// Mitsubishi GX Works2 project: BookEX5_0 ST   PLC: Q13UDV

TYPE DateTime : STRUCT
  Year : INT;
  Month : INT;
  Day : INT;
  WeekDay : INT;
  iHour : INT;
  iMin : INT;
  iSec : INT;
  ms : INT;
END_STRUCT END_TYPE

TYPE Vector : STRUCT
  axisX : REAL;
  axisY : REAL;
  axisZ : REAL;
END_STRUCT END_TYPE

TYPE WordBit : STRUCT
  Data : DWORD;
  Flag : BOOL;
END_STRUCT END_TYPE

// global labels: Global
VAR_GLOBAL
  bVar0 AT M5000 : BOOL;
  abArray0 AT M5010 : ARRAY [0..49] OF BOOL;
  sStr0 AT D5000 : STRING[199];
  sStr1 AT D5100 : STRING[199];
  sStr2 AT D5200 : STRING[199];
  sStr3 AT D5300 : STRING[199];
  sStr4 AT D5400 : STRING[199];
  sStr5 AT D5500 : STRING[199];
  sStr6 AT D5600 : STRING[199];
  sStr7 AT D5700 : STRING[199];
  sStr8 AT D5800 : STRING[199];
  sStr9 AT D5900 : STRING[199];
  iVar0 AT D4500 : INT;
  iVar1 AT D4501 : INT;
  iVar2 AT D4502 : INT;
  iVar3 AT D4503 : INT;
  iVar4 AT D4504 : INT;
  iVar5 AT D4505 : INT;
  iVar6 AT D4506 : INT;
  iVar7 AT D4507 : INT;
  iVar8 AT D4508 : INT;
  iVar9 AT D4509 : INT;
  dVar0 AT D4510 : DINT;
  dVar1 AT D4512 : DINT;
  dVar2 AT D4514 : DINT;
  dVar3 AT D4516 : DINT;
  dVar4 AT D4518 : DINT;
  dVar5 AT D4520 : DINT;
  dVar6 AT D4522 : DINT;
  dVar7 AT D4524 : DINT;
  dVar8 AT D4526 : DINT;
  dVar9 AT D4528 : DINT;
  wVar0 AT D4530 : WORD;
  wVar1 AT D4531 : WORD;
  wVar2 AT D4532 : WORD;
  wVar3 AT D4533 : WORD;
  wVar4 AT D4534 : WORD;
  wVar5 AT D4535 : WORD;
  wVar6 AT D4536 : WORD;
  wVar7 AT D4537 : WORD;
  wVar8 AT D4538 : WORD;
  wVar9 AT D4539 : WORD;
  dwVar0 AT D4540 : DWORD;
  dwVar1 AT D4542 : DWORD;
  dwVar2 AT D4544 : DWORD;
  dwVar3 AT D4546 : DWORD;
  dwVar4 AT D4548 : DWORD;
  dwVar5 AT D4550 : DWORD;
  dwVar6 AT D4552 : DWORD;
  dwVar7 AT D4554 : DWORD;
  dwVar8 AT D4556 : DWORD;
  dwVar9 AT D4558 : DWORD;
  fsVar0 AT D4560 : REAL;
  fsVar1 AT D4562 : REAL;
  fsVar2 AT D4564 : REAL;
  fsVar3 AT D4566 : REAL;
  fsVar4 AT D4568 : REAL;
  fsVar5 AT D4570 : REAL;
  fsVar6 AT D4572 : REAL;
  fsVar7 AT D4574 : REAL;
  fsVar8 AT D4576 : REAL;
  fsVar9 AT D4578 : REAL;
  fdVar0 AT D4580 : LREAL;
  tTime0 AT D4620 : TIME;
  tTime1 AT D4622 : TIME;
  tTime2 AT D4624 : TIME;
  tTime3 AT D4626 : TIME;
  tTime4 AT D4628 : TIME;
  tTime5 AT D4630 : TIME;
  tTime6 AT D4632 : TIME;
  tTime7 AT D4634 : TIME;
  tTime8 AT D4636 : TIME;
  tTime9 AT D4638 : TIME;
  tTime10 AT D4640 : TIME;
  bVar1 AT M5001 : BOOL;
  bVar2 AT M5002 : BOOL;
  bVar3 AT M5003 : BOOL;
  bVar4 AT M5004 : BOOL;
  bVar5 AT M5005 : BOOL;
  bVar6 AT M5006 : BOOL;
  bVar7 AT M5007 : BOOL;
  bVar8 AT M5008 : BOOL;
  bVar9 AT M5009 : BOOL;
  abArray1 AT M5060 : ARRAY [0..49] OF BOOL;
  abArray2 AT M5110 : ARRAY [0..49] OF BOOL;
  abArray3 AT M5160 : ARRAY [0..49] OF BOOL;
  abArray4 AT M5210 : ARRAY [0..49] OF BOOL;
  abArray5 AT M5260 : ARRAY [0..49] OF BOOL;
  abArray6 AT M5310 : ARRAY [0..49] OF BOOL;
  abArray7 AT M5360 : ARRAY [0..49] OF BOOL;
  abArray8 AT M5410 : ARRAY [0..49] OF BOOL;
  abArray9 AT M5460 : ARRAY [0..49] OF BOOL;
  fdVar1 AT D4584 : LREAL;
  fdVar2 AT D4588 : LREAL;
  fdVar3 AT D4592 : LREAL;
  fdVar4 AT D4596 : LREAL;
  fdVar5 AT D4600 : LREAL;
  fdVar6 AT D4604 : LREAL;
  fdVar7 AT D4608 : LREAL;
  fdVar8 AT D4612 : LREAL;
  fdVar9 AT D4616 : LREAL;
  aSendData1 AT D100 : ARRAY [0..9] OF INT;
  aRecvData1 AT D110 : ARRAY [0..9] OF INT;
  aSendData2 AT D120 : ARRAY [0..9] OF INT;
  aRecvData2 AT D130 : ARRAY [0..9] OF INT;
END_VAR
// user libraries (not included): HMI

FUNCTION_BLOCK AllFB
VAR_INPUT
  b_IN1 : BOOL;
  b_IN2 : BOOL;
END_VAR
VAR_OUTPUT
  b_OT : BOOL;
END_VAR
(* structured ladder/FBD written out as ST: instructions are called as NAME(EN, inputs, outputs); _pN, _eN, _tN stand for wires *)
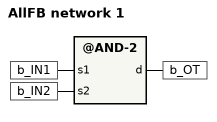
(* network 1 *)
b_OT := @AND-2(b_IN1, b_IN2);
END_FUNCTION_BLOCK

FUNCTION_BLOCK EnFB
VAR_INPUT
  b_IN1 : BOOL;
  b_IN2 : BOOL;
END_VAR
VAR_OUTPUT
  b_OT : BOOL;
END_VAR
(* structured ladder/FBD written out as ST: instructions are called as NAME(EN, inputs, outputs); _pN, _eN, _tN stand for wires *)
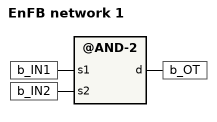
(* network 1 *)
b_OT := @AND-2(b_IN1, b_IN2);
END_FUNCTION_BLOCK

FUNCTION EnFUN
VAR_INPUT
  b_IN1 : BOOL;
  b_IN2 : BOOL;
END_VAR
(* structured ladder/FBD written out as ST: instructions are called as NAME(EN, inputs, outputs); _pN, _eN, _tN stand for wires *)
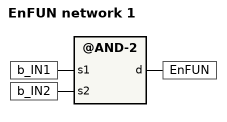
(* network 1 *)
EnFUN := @AND-2(b_IN1, b_IN2);
END_FUNCTION

FUNCTION_BLOCK MacroEnFB
VAR_INPUT
  b_IN1 : BOOL;
  b_IN2 : BOOL;
END_VAR
VAR_OUTPUT
  b_OT : BOOL;
END_VAR
(* structured ladder/FBD written out as ST: instructions are called as NAME(EN, inputs, outputs); _pN, _eN, _tN stand for wires *)
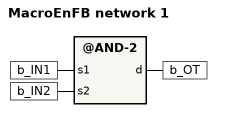
(* network 1 *)
b_OT := @AND-2(b_IN1, b_IN2);
END_FUNCTION_BLOCK

FUNCTION_BLOCK MacroFB
VAR_INPUT
  b_IN1 : BOOL;
  b_IN2 : BOOL;
END_VAR
VAR_OUTPUT
  b_OT : BOOL;
END_VAR
VAR
  ix : INT;
END_VAR
(* structured ladder/FBD written out as ST: instructions are called as NAME(EN, inputs, outputs); _pN, _eN, _tN stand for wires *)
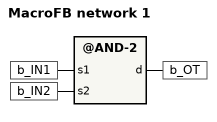
(* network 1 *)
b_OT := @AND-2(b_IN1, b_IN2);
END_FUNCTION_BLOCK

FUNCTION_BLOCK ManEnFB
VAR_INPUT
  b_EN : BOOL;
  b_IN2 : BOOL;
END_VAR
VAR_OUTPUT
  b_OT : BOOL;
END_VAR
VAR
  ix : INT;
END_VAR
VAR_INPUT
  b_IN1 : BOOL;
END_VAR
VAR_OUTPUT
  b_ENO : BOOL;
END_VAR
(* structured ladder/FBD written out as ST: instructions are called as NAME(EN, inputs, outputs); _pN, _eN, _tN stand for wires *)
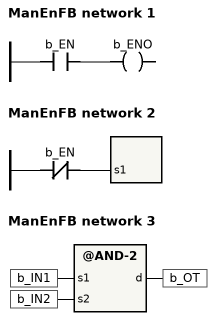
(* network 1 *)
b_ENO := b_EN;
(* network 2 *)
(* element kind 10  <- NOT b_EN *)
(* network 3 *)
b_OT := @AND-2(b_IN1, b_IN2);
END_FUNCTION_BLOCK

FUNCTION_BLOCK NoneFB
VAR_INPUT
  b_IN1 : BOOL;
  b_IN2 : BOOL;
END_VAR
VAR_OUTPUT
  b_OT : BOOL;
END_VAR
(* structured ladder/FBD written out as ST: instructions are called as NAME(EN, inputs, outputs); _pN, _eN, _tN stand for wires *)
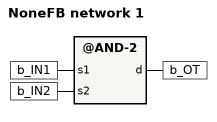
(* network 1 *)
b_OT := @AND-2(b_IN1, b_IN2);
END_FUNCTION_BLOCK

FUNCTION NoneFUN
VAR_INPUT
  b_IN1 : BOOL;
  b_IN2 : BOOL;
END_VAR
(* structured ladder/FBD written out as ST: instructions are called as NAME(EN, inputs, outputs); _pN, _eN, _tN stand for wires *)
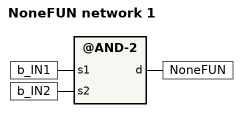
(* network 1 *)
NoneFUN := @AND-2(b_IN1, b_IN2);
END_FUNCTION

PROGRAM 000DataType
VAR
  aBoxNo : ARRAY [0..99] OF INT;
  aStr : ARRAY [0..9] OF STRING[4] := [10('')];
  aStr2 : ARRAY [0..19] OF STRING[32] := [20('')];
  ai박스3 : ARRAY [0..4,0..3,0..2] OF INT;
  aiBox1 : ARRAY [0..4] OF INT;
  aiBox2 : ARRAY [1..5] OF INT;
  ai박스2 : ARRAY [-1..4,1..3] OF INT;
  ix : INT;
  Val1 : INT;
  Val2 : INT;
  Val3 : INT;
  abLable2 : ARRAY [0..4,0..3] OF BOOL;
  abLable1 : ARRAY [0..3] OF BOOL;
  abLabel3 : ARRAY [0..5,0..4,0..3] OF BOOL;
END_VAR
 
FOR ix := 0 TO 99 DO
	aBoxNo[ix] := ix;
END_FOR;
aiBox1[0] := 12;
aiBox1[2] := 34;
aStr[0] := 'ABCDEFG';		(* No Error *)
aStr[1] := '12345678';		(* No Error *)
Val2 := ai박스2[1,1]; 	 
Val3 := 100;
aBoxNo[Val3] := 100;		(* No Error *)
aBoxNo[aBoxNo[aBoxNo[aBoxNo[aBoxNo[Val3]]]]] := 100;
aiBox2 := aiBox1;

Val1 := aBoxNo[55];

bVar0 	:= 1;
bVar1	:= TRUE;
fsVar5	:= E1.0E-5;
fsVar6	:= 1.0E-5;
wVar0	:= 16#FF_FF;
wVar1	:= HFFFF;
aStr2[0]:= 'APP';
aStr2[1]:= '$$';
aStr2[2]:= "$N";
aStr2[3]:= "$n";
aStr2[4]:= "$5C";

MOVP(X1, K3M0, iVar1);

MOVP(X1, K3M0, D40);

DMOVP(X1, 155, dVar0);

DMOVP(X1, 155, D12);

EMOVP(X1, fsVar0, fsVar1);

EDMOVP(X1, 1.23456, fdVar0);
END_PROGRAM

PROGRAM ExCallFB
VAR
  TON_E_1 : TON_E;
  TON_E_2 : TON_E;
  TON_E_3 : TON_E;
  TON_E_4 : TON_E;
END_VAR
 
iVar4 := iVar4 + 1;

TON_E_1.IN := FALSE;
TON_E_1.PT := T#1s;
TON_E_1(EN:=TRUE, IN:=M1);
IF TON_E_1.Q THEN
	TON_E_1(EN:=TRUE, IN:=FALSE);
	iVar1 := iVar1 + 1;
END_IF;
tTime1 := TON_E_1.ET;

TON_E_2(EN:=TRUE, IN:=M1, PT:= T#2s);
IF TON_E_2.Q THEN
	TON_E_2(EN:=TRUE, IN:=FALSE);
	iVar2 := iVar2 + 1;
END_IF;
tTime2 := TON_E_2.ET;

TON_E_3.IN := M1;
TON_E_3.PT := T#3s;
TON_E_3(EN:=TRUE);
IF TON_E_3.Q THEN
	TON_E_3(EN:=TRUE, IN:=FALSE);
	iVar3 := iVar3 + 1;
END_IF;
tTime3 := TON_E_3.ET;

TON_E_4(EN:=TRUE, IN:=M1, PT:= T#2s);
M4 := TON_E_4.Q;
tTime4 := TON_E_4.ET;
IF M4 THEN
	TON_E_4(EN:=TRUE, IN:=FALSE);
	iVar4 := iVar4 + 1;
END_IF;
END_PROGRAM

PROGRAM ExFB
VAR
  NoneFB_1 : NoneFB;
  EnFB_1 : EnFB;
  MacroFB_1 : MacroFB;
  AllFB_1 : AllFB;
  MacroEnFB_1 : MacroEnFB;
  ManEnFB_1 : ManEnFB;
END_VAR
(* structured ladder/FBD written out as ST: instructions are called as NAME(EN, inputs, outputs); _pN, _eN, _tN stand for wires *)
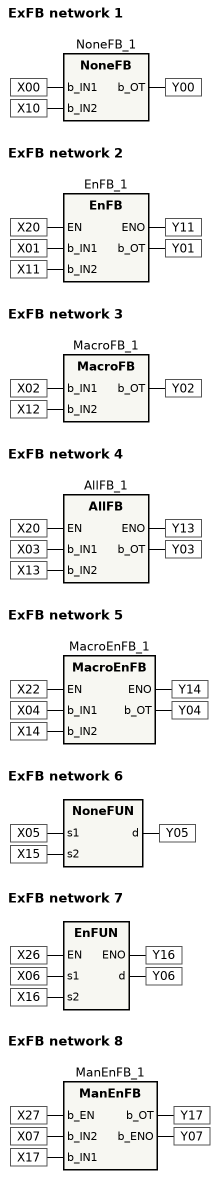
(* network 1 *)
NoneFB_1(b_IN1 := X00, b_IN2 := X10, b_OT => Y00);
(* network 2 *)
EnFB_1(EN := X20, b_IN1 := X01, b_IN2 := X11, ENO => Y11, b_OT => Y01);
(* network 3 *)
MacroFB_1(b_IN1 := X02, b_IN2 := X12, b_OT => Y02);
(* network 4 *)
AllFB_1(EN := X20, b_IN1 := X03, b_IN2 := X13, ENO => Y13, b_OT => Y03);
(* network 5 *)
MacroEnFB_1(EN := X22, b_IN1 := X04, b_IN2 := X14, ENO => Y14, b_OT => Y04);
(* network 6 *)
Y05 := NoneFUN(X05, X15);
(* network 7 *)
_e1 := EnFUN(X26, X06, X16, Y06);
Y16 := _e1;
(* network 8 *)
ManEnFB_1(b_EN := X27, b_IN2 := X07, b_IN1 := X17, b_OT => Y17, b_ENO => Y07);
END_PROGRAM

PROGRAM ExFOR
VAR
  Result1 : BOOL;
  Result2 : BOOL;
END_VAR

iVar4 := 0;
FOR iVar3 := 1 TO 10 BY 1 DO 
	iVar4 := iVar3+iVar4;
END_FOR;

iVar6 := 0;
FOR iVar5 := 10 TO 1 BY -1 DO 
	iVar6 := iVar5+iVar6;
END_FOR;
END_PROGRAM

PROGRAM ExOperator
;
(*기본 연산자*)
iVar0 := iVar1 * iVar2 + iVar3 MOD 16;							(* INT *)
iVar4 := (iVar5 + D0 + iVar6) / 3;
(* iVar0 := dVar1 * iVar2 + iVar3 MOD 16;  데이터형이 틀리면 에러 *)

D0 := iVar1 * D2 + iVar3 MOD 16;
D0 := D1 * (D2+3) / 100;
(* D0 := dVar1 * dVar2 + dVar3 MOD 16;   D0는 INT로 처리함으로 에러 *)

dVar0 := dVar1 * dVar2 / 4 + dVar3 MOD 16;					(* DINT *)
dVar4 := dVar5 / H1000;
(*wVar0 := wVar1 * wVar2 + wVar3 MOD 16;  Bit-string은 일반 연산자 사용시 에러 *)

fsVar0 := fsVar1 + fsVar3 * 2.0;												(* REAL *)
fsVar1 := 2.0  * 3.14 * fsVar5;
fdVar0 := fdVar1 + fdVar2 ** 2.0;

(* sStr0 := sStr0 + "ABC";							String은 일반 연산자 사용시 에러 *)
tTime0 := tTime1+tTime2;															(* Time *)
tTime3 := tTime4 + T#1s;

(*고급 연산자*)
iVar0 := ABS(iVar2 - iVar3);														(* INT *)
dVar0 := ABS(dVar2 - dVar3);													(* DINT *)

fsVar0 := ABS(fsVar1 - fsVar2) + INT_TO_REAL(iVar0);	(* REAL *)
bVar0 := SIN_E (TRUE, fdVar1, fdVar0);
fdVar2 := SQRT((fdVar0 ** 2.0) + (fdVar1 ** 2.0));

(*논리 연산자 *)
bVar0 := bVar1 XOR M0 AND (iVar0 = 100);								(* Bit *)
D1.3 := NOT ( bVar3 AND bVar4);

D0 := D1 AND D2;																				(* WORD *)
wVar1 := wVar1 XOR wVar2;
wVar3 := wVar4 OR H0011;
D3 := D2 OR wVar1;
(* D3 := D2 OR iVar1;  D0는 WORD로  처리함으로 에러 *)

dwVar1 := dwVar1 XOR dwVar2;													(* DWORD *)
dwVar3 := NOT (dwVar4 OR dwVar1) AND H0F0F0F0F;
(* D3 := D2 OR dwVar1;  D0는 WORD로  처리함으로 에러 *)

(*관계연산자*)
bVar0 := bVar1 < bVar2;																	(* Bit *)
bVar0 := ( D0 > 100 ) AND (D0 < 200);											(* INT *)
bVar3 := dVar1 >= 100;																	(* DINT *)
bVar4 := (wVar0 AND H00FF) = 0;												(* WORD *)
bVar4 := wVar1 = H0100;
bVar4 := wVar2 > H0100;
bVar5 := (dwVar0 AND H00FF) <> 0;											(* DWORD *)
bVar6 := dwVar1 <> HFFFFFFFF;
IF D0 = 100 THEN bVar1 := TRUE; ELSE bVar1 := FALSE; END_IF;
bVar7 := tTime0 < tTime1;																(* Time *)
bVar7 := tTime2 > T#200s;
END_PROGRAM

PROGRAM ExREPEAT
VAR
  Result1 : BOOL;
  Result2 : BOOL;
END_VAR

iVar6 := 0;
iVar5 := 1;
REPEAT
	iVar6 := iVar5 + iVar6;
	iVar5 := iVar5 + 1;
	UNTIL iVar5 > 10  
END_REPEAT;
END_PROGRAM

PROGRAM ExST
VAR
  ix : INT;
END_VAR
VAR CONSTANT
  MaxCnt : INT := 100;
END_VAR
VAR
  aaa : ARRAY [0..4,0..4,0..4] OF INT;
  aDT0 : ARRAY [0..2] OF DateTime;
  aDT1 : ARRAY [0..2] OF DateTime;
  DT0 : DateTime;
  DT1 : DateTime;
  aiClass1 : ARRAY [0..9] OF INT;
  aiClass2 : ARRAY [0..9] OF INT;
  Res1 : INT;
  Res2 : INT;
  Res3 : INT;
  Res4 : INT;
END_VAR

(* ST 샘플 츠로그램 *)
wVar1	:= H1234;
dwVar1	:= 12345678;

bVar1	:= BCD_TO_DINT_E(TRUE, wVar1, dVar1);
dVar2	:= BCD_TO_DINT(wVar1);

bVar2	:= ADD_E(TRUE, iVar1, iVar2, iVar3, iVar4, iVar5);
iVar5		:= iVar1 + iVar2 + iVar3 + iVar4;

IF NOT (bVar1 AND NOT bVar2 AND M0) THEN
	bVar2	:= TRUE;
ELSE
	bVar2	:= FALSE;
END_IF;

fbDispHMI(Bit0 := bVar1, Bit1 := bVar2); (* HMI표시를 위한 함수 *)
bVar4	:= fbDispHMI.Data0;


iVar0		:= D10 - 123;

IF iVar0 > 0 THEN
	bVar0	:= TRUE;
ELSE
	bVar1	:= FALSE;
END_IF;

WHILE FunPOU(iVar0) DO
	iVar0		:= iVar0 - 1;
END_WHILE;

bFlag 	:= FunPOU(iVar0 + 1);
fbPOU_1(In0 := iVar0 + 1, Out0 := iVar1);



WHILE bVar0 DO
	iVar0		:= iVar0 - 1;
	IF iVar0 > 100 THEN
		bVar0	:= TRUE;
	ELSE
		IF iVar0 > 50 THEN
			iVar1	:= iVar1 + 1;
		END_IF;
	END_IF;
END_WHILE;




(* 대입문*)
iVar1 			:= iVar2;					iVar3 := 0;
iVar4 			:= iVar4 + 1;
D1 				:= iVar1;
wVar2 		:= INT_TO_WORD(iVar3);
sStr1 			:= 'abc';
sStr2			:= "Apple";

IF LDP(TRUE, M0) THEN
	iVar5 := aiClass2[3];
	iVar7 := DT1.Month;
	aiClass1[3] := 3;
	aDT0[1].Month := 12;
	aiClass2 := aiClass1;
	DT1 := aDT0[1];
	iVar6 := aiClass2[3];
	iVar8 := DT1.Month;
END_IF;

(* IF ... THEN *)
IF M0 THEN
	Y0 := TRUE;
END_IF;

(* IF ... ELSE *)
IF M0 THEN
	Y0 := TRUE;
ELSE
	Y0 := FALSE;
END_IF;

(* IF ... ELSIF *)
IF M0 THEN
	Y0 := TRUE;
ELSIF M1 THEN
	Y1 := TRUE;
ELSIF M2 THEN
	Y2 := TRUE;
END_IF;

(* CASE *)
IF (iVar0 = 0) THEN
	Res1 := iVar0 + 5;
ELSIF(iVar0 = 1) THEN
	Res1 := iVar0 + 10;
ELSIF(iVar0 = 2) THEN
	Res1 := iVar0 + 15;
ELSIF(iVar0 = 3) THEN
	Res1 := iVar0 + 20;
ELSIF(iVar0 = 4) THEN
	Res1 := iVar0 + 25;
ELSIF(iVar0 = 5) THEN
	Res1 := iVar0 + 30;
ELSE
	Res1 := 0;
END_IF;

CASE iVar0 OF
 	0 : 	Res2 := iVar0 + 5;
	1 :	Res2 := iVar0 + 10;
	2 :	Res2 := iVar0 + 15;
	3 :	Res2 := iVar0 + 20;
	4 :	Res2 := iVar0 + 25;
	5 :	Res2 := iVar0 + 30;
	ELSE
			Res2 := 0;
END_CASE;

CASE iVar0 OF
 	0,1,2 : Res3 := (iVar0+1) * 5 + iVar0;
	3..5   :	Res3 := (iVar0+1) * 5 + iVar0;;
	ELSE
			Res3 := 0;
END_CASE;

(* CASE *)
CASE D0 OF
	1 : 	Y0 := TRUE;
	2 : 	Y1 := TRUE;
	3 : 	Y2 := TRUE;
	ELSE
			Y3 := TRUE;
END_CASE;

CASE D0 OF
	1 : 	Y0 := TRUE;
	2 : 	Y1 := TRUE;
	3 : 	Y2 := TRUE;
END_CASE;

(* FOR *)
FOR D0 := 0 TO 100 BY 1 DO 
	D1 := D1 + 1;
END_FOR;

FOR D0 := 0 TO 100 DO 
	D1 := D1 + 1;
END_FOR;

FOR D0 := 100 TO 0 BY -1 DO 
	D1 := D1 + 1;
END_FOR;

(* WHILE *)
iVar3 := 0;
WHILE iVar3 < 100 DO 
	iVar3 := iVar3 +1;
END_WHILE;

(* REPEAT *)
iVar4 := 0;
REPEAT 
	iVar4 := iVar4 +1;
	UNTIL iVar4 < 100 
END_REPEAT;

(* RETUEN *)
IF M0 THEN
	RETURN; 
END_IF;

(* EXIT *)
FOR D0 := 0 TO 100 DO 
	IF D0 = 30 THEN
		EXIT;
	END_IF;
END_FOR;

RETURN;

IF (iVar1 = 0) AND (iVar3 = 2) THEN
	iVar2 := 123;
ELSIF X0 AND X1 THEN
	iVar2 := 321;
ELSIF X0 OR X1 THEN
	iVar2 := 456;
ELSE
	iVar2 := 567;
END_IF;


(* IF문 계층 Test *)
IF iVar1 = 0 THEN
	iVar2 := 0;
	IF iVar1 = 0 THEN
		iVar2 := 1;
		IF iVar1 = 0 THEN
			iVar2 := 2;
			IF iVar1 = 0 THEN
				iVar2 := 3;
				IF iVar1 = 0 THEN
					iVar2 := 4;
					IF iVar1 = 0 THEN
						iVar2 := 5;
						IF iVar1 = 0 THEN
							iVar2 := 6;
							IF iVar1 = 0 THEN
								iVar2 := 7;
								IF iVar1 = 0 THEN
									iVar2 := 8;
									IF iVar1 = 0 THEN
										iVar2 := 9;
										IF iVar1 = 0 THEN
											iVar2 := 10;
											IF iVar1 = 0 THEN
												iVar2 := 11;
												IF iVar1 = 0 THEN
													iVar2 := 12;
													IF iVar1 = 0 THEN
														iVar2 := 13;
														IF iVar1 = 0 THEN
															iVar2 := 14;
															IF iVar1 = 0 THEN
																iVar2 := 15;
																IF iVar1 = 0 THEN
																	iVar2 := 16;
																	IF iVar1 = 0 THEN
																		iVar2 := 17;
																		IF iVar1 = 0 THEN
																			iVar2 := 18;
																		END_IF;
																	END_IF;
																END_IF;
															END_IF;
														END_IF;
													END_IF;
												END_IF;
											END_IF;
										END_IF;
									END_IF;
								END_IF;
							END_IF;
						END_IF;
					END_IF;
				END_IF;
			END_IF;
		END_IF;
	END_IF;
END_IF;
END_PROGRAM

PROGRAM ExWHILE
VAR
  Result1 : BOOL;
  Result2 : BOOL;
END_VAR

iVar6 := 0;
iVar5 := 1;
WHILE iVar5 <= 10 DO 
	iVar6 := iVar5 + iVar6;
	iVar5 := iVar5 + 1;
END_WHILE;
END_PROGRAM

PROGRAM ExEXIT
;

iVar6	:= 0;
FOR iVar5 := 1 TO 10 DO 
	iVar6	:= iVar5 + iVar6;
	iVar3	:= 0;
	FOR iVar4 := 0 TO 10 DO
		iVar3	:= iVar4 + iVar3;
		IF iVar4 = 5 THEN
			EXIT;
		END_IF;
	END_FOR;
END_FOR;
END_PROGRAM
